FUNCTION_BLOCK necessidade2Equipamentos (* Composite Function Block Type *)
  (* Standard: 61499-2 *)
  (* Version 0.0, 27/02/2026, template *)
  PACKAGE Hidryco.HidrycoLib;
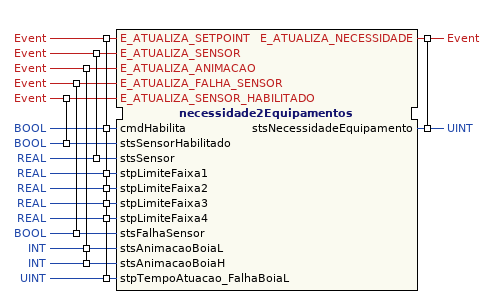
  EVENT_INPUT
    E_ATUALIZA_SETPOINT WITH stpLimiteFaixa1, stpLimiteFaixa2, stpLimiteFaixa3, stpLimiteFaixa4, stpTempoAtuacao_FalhaBoiaL, cmdHabilita;
    E_ATUALIZA_SENSOR WITH stsSensor;
    E_ATUALIZA_ANIMACAO WITH stsAnimacaoBoiaL, stsAnimacaoBoiaH;
    E_ATUALIZA_FALHA_SENSOR WITH stsFalhaSensor;
    E_ATUALIZA_SENSOR_HABILITADO WITH stsSensorHabilitado;
  END_EVENT
  EVENT_OUTPUT
    E_ATUALIZA_NECESSIDADE WITH stsNecessidadeEquipamento;
  END_EVENT
  VAR_INPUT
    cmdHabilita : BOOL;
    stsSensorHabilitado : BOOL;
    stsSensor : REAL;
    stpLimiteFaixa1 : REAL;
    stpLimiteFaixa2 : REAL;
    stpLimiteFaixa3 : REAL;
    stpLimiteFaixa4 : REAL;
    stsFalhaSensor : BOOL;
    stsAnimacaoBoiaL : INT;
    stsAnimacaoBoiaH : INT;
    stpTempoAtuacao_FalhaBoiaL : UINT; (* Tempo para equipamento ficar ligado quando bater na boia H e a boia L estiver em falha *)
  END_VAR
  VAR_OUTPUT
    stsNecessidadeEquipamento : UINT;
  END_VAR
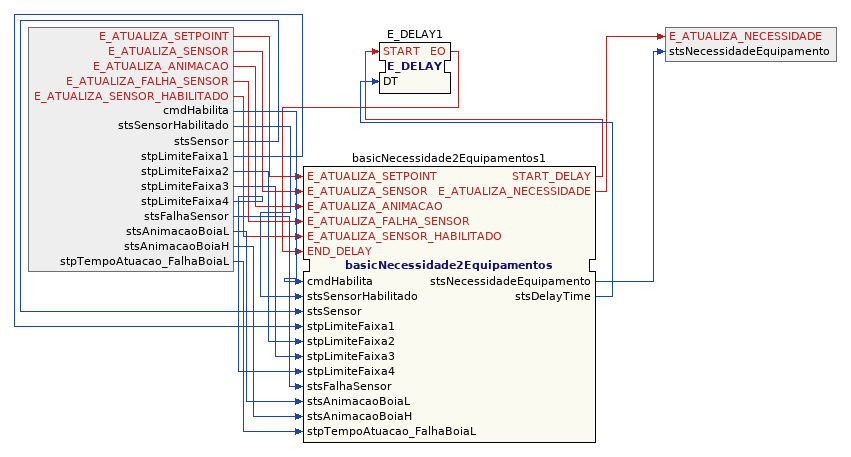
  FBS
    basicNecessidade2Equipamentos1 : basicNecessidade2Equipamentos;
    E_DELAY1 : E_DELAY;
  END_FBS
  EVENT_CONNECTIONS
    E_ATUALIZA_FALHA_SENSOR TO basicNecessidade2Equipamentos1.E_ATUALIZA_FALHA_SENSOR;
    E_ATUALIZA_ANIMACAO TO basicNecessidade2Equipamentos1.E_ATUALIZA_ANIMACAO;
    E_ATUALIZA_SENSOR TO basicNecessidade2Equipamentos1.E_ATUALIZA_SENSOR;
    E_ATUALIZA_SETPOINT TO basicNecessidade2Equipamentos1.E_ATUALIZA_SETPOINT;
    basicNecessidade2Equipamentos1.E_ATUALIZA_NECESSIDADE TO E_ATUALIZA_NECESSIDADE;
    basicNecessidade2Equipamentos1.START_DELAY TO E_DELAY1.START;
    E_DELAY1.EO TO basicNecessidade2Equipamentos1.END_DELAY;
    E_ATUALIZA_SENSOR_HABILITADO TO basicNecessidade2Equipamentos1.E_ATUALIZA_SENSOR_HABILITADO;
  END_CONNECTIONS
  DATA_CONNECTIONS
    stsSensor TO basicNecessidade2Equipamentos1.stsSensor;
    stpLimiteFaixa1 TO basicNecessidade2Equipamentos1.stpLimiteFaixa1;
    stpLimiteFaixa2 TO basicNecessidade2Equipamentos1.stpLimiteFaixa2;
    stpLimiteFaixa3 TO basicNecessidade2Equipamentos1.stpLimiteFaixa3;
    stpLimiteFaixa4 TO basicNecessidade2Equipamentos1.stpLimiteFaixa4;
    stsFalhaSensor TO basicNecessidade2Equipamentos1.stsFalhaSensor;
    stsAnimacaoBoiaL TO basicNecessidade2Equipamentos1.stsAnimacaoBoiaL;
    stsAnimacaoBoiaH TO basicNecessidade2Equipamentos1.stsAnimacaoBoiaH;
    stpTempoAtuacao_FalhaBoiaL TO basicNecessidade2Equipamentos1.stpTempoAtuacao_FalhaBoiaL;
    basicNecessidade2Equipamentos1.stsNecessidadeEquipamento TO stsNecessidadeEquipamento;
    basicNecessidade2Equipamentos1.stsDelayTime TO E_DELAY1.DT;
    cmdHabilita TO basicNecessidade2Equipamentos1.cmdHabilita;
    stsSensorHabilitado TO basicNecessidade2Equipamentos1.stsSensorHabilitado;
  END_CONNECTIONS
END_FUNCTION_BLOCK
